FUNCTION_BLOCK FB_Scale
VAR_INPUT
	X_MIN: REAL;
	X_MAX: REAL;
	Y_MIN: REAL;
	Y_MAX: REAL;
	IN_VALUE: REAL;
END_VAR
VAR_OUTPUT
	OUT_VALUE: REAL;
END_VAR
VAR
	a: REAL;
END_VAR

a := (Y_MAX - Y_MIN) / (X_MAX - X_MIN);
OUT_VALUE := a*(IN_VALUE-X_MIN) + Y_MIN;

END_FUNCTION_BLOCK

(* stored: Version 1.1.0.1, ProductVersion 3.1.4024.4
   POU FB_Scale: Id {f12285d5-1b19-44ea-a3f3-a9cc10e59d5d}, SpecialFunc None *)
